FUNCTION_BLOCK FB_UAgetNameSpaceIndexMock_success IMPLEMENTS I_OPCUA_GetNameSpaceIndex
VAR_INPUT
END_VAR
VAR_OUTPUT
END_VAR
VAR
END_VAR

{warning 'add method implementation '}
METHOD start : BOOL
VAR_INPUT
	Execute	: BOOL;
	ConnectionHdl	: DWORD;
	NamespaceUri	: STRING(MAX_STRING_LENGTH);
	Timeout	: TIME := DEFAULT_ADS_TIMEOUT;
END_VAR
VAR_OUTPUT
	NamespaceIndex	: UINT;
	Done	: BOOL;
	Busy	: BOOL;
	Error	: BOOL;
	ErrorID	: DWORD;
END_VAR
IF execute THEN
	done := TRUE;
END_IF
END_METHOD

END_FUNCTION_BLOCK

(* stored: Version 1.1.0.1, ProductVersion 3.1.4024.9
   POU FB_UAgetNameSpaceIndexMock_success: Id {1dff67b7-b8b7-404b-8228-95edcb450714}, SpecialFunc None
   Method start: Id {113eaf49-9c02-4d40-be9e-146956ae69ea} *)
